// TIA Portal V19 export
FUNCTION_BLOCK "UnsupportedVersion_FB"   // FB, LAD
// stored: SetENOAutomatically false
BEGIN
END_FUNCTION_BLOCK
